FUNCTION_BLOCK FB_LT_UINT (* UINT Comparison *)
  (* Standard: 61499-1-D.1; Classification: Math; Function: Comparison *)
  (* Version 0.0, 2006-04-13, JHC, Holobloc Inc *)
  (* Compiler header: package fb.rt.math; *)
  (* Compiler classdef: class FB_GT_REAL extends FBFunction2 *)
  (* Compiler Java Sun JDK 1.5.0 *)
  (* Compiler Java IBM VisualAge 3.0 *)
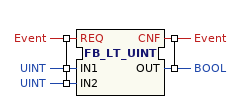
  EVENT_INPUT
    REQ WITH IN1, IN2;
  END_EVENT
  EVENT_OUTPUT
    CNF WITH OUT;
  END_EVENT
  VAR_INPUT
    IN1 : UINT;
    IN2 : UINT;
  END_VAR
  VAR_OUTPUT
    OUT : BOOL; (* IN1>IN2 *)
  END_VAR
END_FUNCTION_BLOCK
